{attribute 'qualified_only'}
VAR_GLOBAL CONSTANT
	// size of the observer array
	cMaxObservers		: INT := 10;	
END_VAR

(* stored: Version 1.1.0.1, ProductVersion 3.1.4022.10
   GVL Param: Id {2ce1f4ec-8da9-48ea-8aa2-bcb508c095b0}, ParameterList True *)
